Universal Robots PolyScope program: CRISTIAN.urp

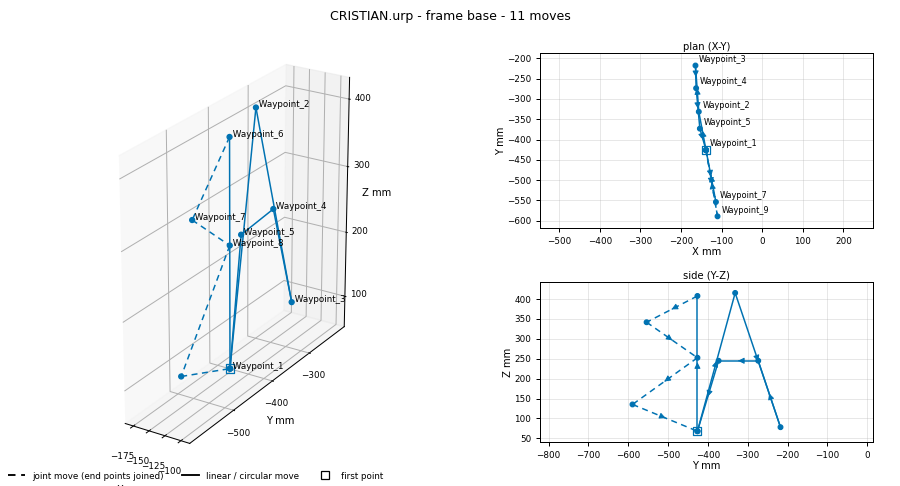
[picture p0: tool path of CRISTIAN.urp in frame base, 11 of 11 moves have a stored position in this frame; points joined in program order, loops and branches not executed]
Program letras (installation=default directory=/ursim/programs createdIn=3.15.8.106339 lastSavedIn=3.15.8.106339 robotSerialNumber=2018359999)
Calibrated DH parameters: a=[0, -0.425, -0.39225, 0, 0, 0]; d=[0.089159, 0, 0, 0.10915, 0.09465, 0.0823]; alpha=[1.570796, 0, 0, 1.570796, -1.570796, 0]; deltaTheta=[0, 0, 0, 0, 0, 0]
Robot Program (runOnlyOnce=false)
  Popup Message (haltProgram=false message=Se va a simular letra A y B inputType=Text)
  'Alejandro Bello'
  MoveL speed 250 mm/s, acceleration 1200 mm/s^2 (useActiveTCP=true) feature=Base
    Waypoint Waypoint_1: TCP in base x=-138.357 y=-426.232 z=68.074 mm, rx=0.0843 ry=-1.5926 rz=0.0533 rad; joints [-82.705, -111.271, -127.029, -91.067, 2.677, -301.673] deg
    Waypoint Waypoint_2: TCP in base x=-156.212 y=-331.504 z=415.273 mm, rx=0.0843 ry=-1.5926 rz=0.0533 rad; joints [-83.744, -69.724, -111.186, -131.932, 1.86, -318.211] deg
    Waypoint Waypoint_3: TCP in base x=-164.403 y=-217.655 z=78.154 mm, rx=0.0843 ry=-1.5926 rz=0.0533 rad; joints [-82.517, -86.78, -156.497, -88.02, 2.84, -299.741] deg
    Waypoint Waypoint_4: TCP in base x=-162.751 y=-273.552 z=244.952 mm, rx=0.0843 ry=-1.5926 rz=0.0533 rad; joints [-83.785, -66.689, -138.89, -106.312, 1.832, -319.162] deg
    Waypoint Waypoint_5: TCP in base x=-153.573 y=-373.13 z=244.952 mm, rx=0.0843 ry=-1.5926 rz=0.0533 rad; joints [-84.051, -82.914, -129.39, -92.762, 1.666, -325.991] deg
    Waypoint Waypoint_1: TCP in base x=-138.357 y=-426.232 z=68.074 mm, rx=0.0843 ry=-1.5926 rz=0.0533 rad; joints [-82.705, -111.271, -127.029, -91.067, 2.677, -301.673] deg
    Waypoint Waypoint_6: TCP in base x=-138.357 y=-426.232 z=407.673 mm, rx=0.0843 ry=-1.5926 rz=0.0533 rad; joints [-82.705, -85.771, -97.434, -146.163, 2.677, -301.673] deg
    MoveJ speed 60 deg/s, acceleration 80 deg/s^2 (useActiveTCP=true)
      Waypoint Waypoint_7: motionParameters(blendRadius=0.1); TCP in base x=-114.015 y=-553.931 z=341.675 mm, rx=0.0843 ry=-1.5926 rz=0.0533 rad; joints [-81.86, -105.399, -84.646, -146.526, 3.432, -294.46] deg
      Waypoint Waypoint_8: TCP in base x=-138.357 y=-426.232 z=252.475 mm, rx=0.0843 ry=-1.5926 rz=0.0533 rad; joints [-82.705, -91.46, -115.551, -122.357, 2.677, -301.673] deg
      Waypoint Waypoint_9: motionParameters(blendRadius=0.1); TCP in base x=-110.019 y=-589.305 z=135.276 mm, rx=0.0843 ry=-1.5926 rz=0.0533 rad; joints [-81.965, -120.677, -95.418, -119.758, 3.335, -295.18] deg
      Waypoint Waypoint_10: TCP in base x=-138.357 y=-426.232 z=68.074 mm, rx=0.0843 ry=-1.5926 rz=0.0533 rad; joints [-82.705, -111.271, -127.029, -91.067, 2.677, -301.673] deg
